(* IEC 61131-3 sources: RL_MAR/experiments/comparison/autoplc/results/gpt-4o_20260511_211137/med_63, 1 file *)

(* ---- med_63_3.st ---- *)
FUNCTION_BLOCK Automated_Parking_Controller
VAR_INPUT
    EntryGateSensor : BOOL; (* Sensor input for entry gate *)
    ExitGateSensor : BOOL; (* Sensor input for exit gate *)
    CarDetected : BOOL; (* Sensor input for car detection *)
END_VAR
VAR_OUTPUT
    ParkingSpaceNumber : INT := 0; (* Allocated parking space number *)
    RetrievalInProgress : BOOL := FALSE; (* Flag for car retrieval in progress *)
END_VAR
VAR
    ParkingSpaces : ARRAY[1..100] OF BOOL; (* Parking space status: TRUE=Occupied, FALSE=Available *)
    i : INT; (* Loop counter *)
    CarSpaceNumber : INT; (* Space number for car retrieval *)
END_VAR

(* Initialization *)
FOR i := 1 TO 100 DO
    ParkingSpaces[i] := FALSE; (* Initialize all parking spaces to available *)
END_FOR

(* Entry Gate Management *)
IF EntryGateSensor AND NOT RetrievalInProgress THEN
    FOR i := 1 TO 100 DO
        IF NOT ParkingSpaces[i] THEN
            ParkingSpaces[i] := TRUE; (* Mark space as occupied *)
            ParkingSpaceNumber := i; (* Output the allocated space number *)
            EXIT; (* Exit the loop once a space is allocated *)
        END_IF
    END_FOR
END_IF

(* Exit Gate Management *)
IF ExitGateSensor THEN
    IF ParkingSpaceNumber > 0 THEN
        ParkingSpaces[ParkingSpaceNumber] := FALSE; (* Mark the space as available *)
        ParkingSpaceNumber := 0; (* Reset the parking space number *)
    END_IF
END_IF

(* Car Retrieval Management *)
IF CarDetected THEN
    RetrievalInProgress := TRUE;
    CarSpaceNumber := ParkingSpaceNumber; (* Store the current parking space number for retrieval *)
    IF MoveCarToExitGate(SpaceNumber := CarSpaceNumber) THEN
        ParkingSpaces[CarSpaceNumber] := FALSE; (* Mark the space as available after retrieval *)
        ParkingSpaceNumber := 0; (* Reset the parking space number *)
        RetrievalInProgress := FALSE; (* Reset retrieval in progress flag *)
    END_IF
END_IF

END_FUNCTION_BLOCK

FUNCTION MoveCarToExitGate : BOOL
VAR_INPUT
    SpaceNumber : INT; (* The parking space number from which the car is to be moved *)
END_VAR
VAR
    MovementComplete : BOOL := FALSE; (* Flag to indicate if the movement is complete *)
END_VAR

(* Simulate car movement logic *)
(* Assume some logic here that moves the car from the given space to the exit gate *)
(* For simplicity, we assume the movement is always successful *)
MovementComplete := TRUE;

(* Return the status of the car movement *)
MoveCarToExitGate := MovementComplete;

END_FUNCTION
